FUNCTION F_PBTrigger : BOOL
VAR_INPUT
    Input : BOOL;
END_VAR
VAR
    Trigger  : R_TRIG;
END_VAR

Trigger(CLK:=Input);

F_PBTrigger := Trigger.Q;

END_FUNCTION

(* stored: Version 1.1.0.1, ProductVersion 3.1.4024.11
   POU F_PBTrigger: Id {71e15ad6-d3c2-4fee-819c-500531ea5599}, SpecialFunc None *)
